TYPE MethodStatus :
STRUCT
	Busy : BIT;
	Error: BIT;
	ErrorID : UDINT;
END_STRUCT
END_TYPE

(* stored: Version 1.1.0.1, ProductVersion 3.1.4024.12
   DUT MethodStatus: Id {f6843048-443c-40db-a5ba-900b15fd3b03} *)
